{attribute 'pack_mode' := '1'}
(* At least one of these components must change for each new
   message sent. 
 *)
TYPE MessageID :
STRUCT
	lowUUID: LINT;    (* Low part of UUID or other unique host identity. *)
	highUUID: LINT;   (* High part of UUID. *)
	dtime: DINT;      (* Time of day in milliseconds. *)
	sequence: DINT;   (* Message sequence number. *)
END_STRUCT
END_TYPE

(* stored: Version 1.1.0.1, ProductVersion 3.1.4022.12
   DUT MessageID: Id {15edb5c5-37c9-47e4-b3b6-3b2b16b8564f} *)
